Fanuc KAREL source: CALL_PROG.kl

PROGRAM T
%NOLOCKGROUP
VAR
 v0 : STRING[40]
 v1 : INTEGER
BEGIN
 CALL_PROG(v0, v1)
END T
